PROGRAM PRG_LVCP1_Group6
VAR
    // Function Block Instance
    fbContactor: FB_ContactorControl;

    // Contactor 1 IO Structure  
    stContactor_IO: ST_ContactorIO;
    
    // Başlangıç konfigürasyonu için flag
    bContactorInitDone: BOOL := FALSE;
    bCapacitorInitDone: BOOL := FALSE;	
END_VAR



	M_Contactor();
	
	M_Capacitor();

METHOD M_Capacitor : BOOL
VAR
    nGroupIndex : INT;
END_VAR

nGroupIndex := 5;  // Grup 6 için index

IF NOT bCapacitorInitDone THEN
    // Grup 6 değerlerini ata
    GVL_LVCP1.astCompensationGroups[nGroupIndex].rPower := 25.0;
    GVL_LVCP1.astCompensationGroups[nGroupIndex].rVoltage := 450.0;
    GVL_LVCP1.astCompensationGroups[nGroupIndex].nQuantity := 3;
    GVL_LVCP1.astCompensationGroups[nGroupIndex].sTagPrefix := '+EP6-31C1';
    GVL_LVCP1.astCompensationGroups[nGroupIndex].sProductCode := 'ENT.CXD-450-25';
    
    bCapacitorInitDone := TRUE;
END_IF

// Grup 6 aktif durumu
GVL_LVCP1.abGroupActive[nGroupIndex] := stContactor_IO.bFeedback;

M_Capacitor := TRUE;
END_METHOD

METHOD M_Contactor : BOOL
VAR_INPUT
END_VAR
IF NOT bContactorInitDone THEN
    // Konfigürasyon parametreleri
    GVL_LVCP1.stGroup6_ContactorHMI.stConfig.sProjectCode := '+EP6-30K1';
    GVL_LVCP1.stGroup6_ContactorHMI.stConfig.sProductCode := 'SCH LC1G265LSEA';
    GVL_LVCP1.stGroup6_ContactorHMI.stConfig.rRatedCurrent := 265.0;
    GVL_LVCP1.stGroup6_ContactorHMI.stConfig.rRatedVoltage := 1000.0;
    GVL_LVCP1.stGroup6_ContactorHMI.stConfig.nPhaseCount := 3;
    GVL_LVCP1.stGroup6_ContactorHMI.stConfig.tFeedbackDelay := T#500MS;
    GVL_LVCP1.stGroup6_ContactorHMI.stConfig.tWeldedDelay := T#2S;
    GVL_LVCP1.stGroup6_ContactorHMI.stConfig.dwOperationLimit := 100000;
    
    // Başlangıç bakım sayacı
    GVL_LVCP1.stGroup6_ContactorHMI.stStatistics.dwRemainingOperations := GVL_LVCP1.stGroup6_ContactorHMI.stConfig.dwOperationLimit;
    
    bContactorInitDone := TRUE;
END_IF

// Function Block Çağrısı
fbContactor(
    // Fiziksel Girişler
    bFeedback := stContactor_IO.bFeedback,
    bPLCControl := stContactor_IO.bPLCControl,
    
    // Güvenlik Girişleri
    bSafetyLoop := GVL_Alarm.bSafetyLoop,
    bInterlock := FALSE,
    
    // Sistem Girişleri
    bMasterReset := GVL_Alarm.bMasterReset,
    
    // HMI Bağlantısı
    stHMI := GVL_LVCP1.stGroup6_ContactorHMI,
    
    // Fiziksel Çıkış
    bOutput => stContactor_IO.bOutput
);

M_Contactor := TRUE;
END_METHOD

END_PROGRAM

(* stored: Version 1.1.0.1, ProductVersion 3.1.4024.15
   POU PRG_LVCP1_Group6: Id {51bc4a9a-d5dd-4000-bc01-a937b5392aca}, SpecialFunc None
   Method M_Capacitor: Id {4a8c0539-d321-4982-8ea2-6bef23ff9f97}
   Method M_Contactor: Id {0a2d14e8-6239-4e10-962c-30b601c7b4c7} *)
